(* CODESYS project project1.project

Project tree, tasks and I/O mapping:
  Device : CODESYS Control Win V3, 3S - Smart Software Solutions GmbH, order no. 305021, version 3.5.10.30
    application Application
      libraries: Standard, * (System)
      task MainTask (cyclic, interval t#20ms, priority 1) calls PLC_PRG
      program PLC_PRG [ST]
*)

// Device/Application/PLC_PRG
PROGRAM PLC_PRG
VAR
END_VAR

END_PROGRAM
